Fanuc KAREL source: V_CSAPI_SAVEDATA.kl

PROGRAM T
%NOLOCKGROUP
VAR
 v0 : STRING[40]
 v1 : INTEGER
BEGIN
 V_CSAPI_SAVEDATA(v0, v1)
END T
